(* PLC project SingleResponsibility.project, CODESYS CODESYS V3.5 SP10 Patch 4 *)
(* stored: creationDateTime 2017-07-22T20:32:32.9692432, modificationDateTime 2017-06-30T11:24:00.4798052 *)

INTERFACE IEStoppable
METHOD executeEStop
END_METHOD
END_INTERFACE

INTERFACE IRunnable
METHOD run
END_METHOD
END_INTERFACE

INTERFACE IStoppable
METHOD stop
END_METHOD
END_INTERFACE

INTERFACE IEdge
METHOD isRising : BOOL
END_METHOD
METHOD isFalling : BOOL
END_METHOD
END_INTERFACE

INTERFACE ISensor
METHOD isOccupied : BOOL
END_METHOD
METHOD isFree : BOOL
END_METHOD
END_INTERFACE

INTERFACE IReciverInterface
METHOD readExtCondition2Rec : IReciverInterface
  VAR_INPUT
    receiveCondition : BOOL;  (* condition 4 ready to receive *)
  END_VAR
END_METHOD
METHOD isReceiving : BOOL
END_METHOD
END_INTERFACE

INTERFACE ISenderInterface
METHOD readExtCondition2Snd : ISenderInterface
  VAR_INPUT
    sendCondition : BOOL;  (* condition 4 ready 2 send *)
  END_VAR
END_METHOD
METHOD isSending : BOOL
END_METHOD
END_INTERFACE

INTERFACE ISmema
METHOD setCondition
  VAR_INPUT
    smemaCondition : BOOL;  (* must be ture to activate the smema interface *)
  END_VAR
END_METHOD
METHOD isTransferActive : BOOL
END_METHOD
END_INTERFACE

INTERFACE ITwoStageLinearDrive
METHOD fastForward
END_METHOD
METHOD forward
END_METHOD
METHOD fastBackward
END_METHOD
METHOD backward
END_METHOD
END_INTERFACE

INTERFACE ITwoStageRotationDrive
METHOD fastClockwise
END_METHOD
METHOD clockwise
END_METHOD
METHOD fastCounterClockwise
END_METHOD
METHOD counterClockwise
END_METHOD
END_INTERFACE

INTERFACE IMachineState
METHOD isMachineInInitMode : BOOL
END_METHOD
METHOD isMachineInIdle : BOOL
END_METHOD
METHOD isMachineInSetup : BOOL
END_METHOD
METHOD isMachineInAutomatic : BOOL
END_METHOD
METHOD isMachineInEstop : BOOL
END_METHOD
END_INTERFACE

FUNCTION_BLOCK DebouncedDigitalSensor IMPLEMENTS ISensor, IEdge
  VAR
    diSensor : REFERENCE TO BOOL;  (* reference to the digital input *)
    maskOccupied : BOOL;  (* mask for the state occupied *)
    debouncer : TON;  (* ton to debounce the sensor signal *)
    debounceTime : TIME;  (* debounce time *)
    state : BOOL;  (* sensor state *)
  END_VAR

            
          

METHOD isOccupied : BOOL
                  isOccupied := isSensorInState(state := THIS^.maskOccupied);
                
END_METHOD

METHOD isFree : BOOL
                  isFree := isSensorInState(state := (NOT THIS^.maskOccupied));
                
END_METHOD

METHOD isRising : BOOL
                  isRising 	:= (THIS^.isOccupied() AND (NOT THIS^.state));
THIS^.updateState();
                
END_METHOD

METHOD isFalling : BOOL
                  isFalling 	:= (THIS^.isFree() AND THIS^.state);
THIS^.updateState();
                
END_METHOD

METHOD FB_INIT
  VAR_INPUT
    bInitRetains : BOOL;  (* initializing of retain-variable *)
    bInCopyCode : BOOL;  (* instance is copied to copy-code *)
    diSensor : REFERENCE TO BOOL;  (* reference to the digital input *)
    maskOccupied : BOOL;  (* mask for the state occupied *)
  END_VAR
                  THIS^.diSensor		REF=diSensor; 
THIS^.maskOccupied	:= maskOccupied;
THIS^.debounceTime	:= T#30ms;
THIS^.state			:= (THIS^.diSensor = THIS^.maskOccupied);
                
END_METHOD

METHOD isSensorInState : BOOL
  VAR_INPUT
    state : BOOL;  (* requeseted sensor state *)
  END_VAR
                  THIS^.debouncer(IN := (THIS^.diSensor = state), PT := THIS^.debounceTime, Q => isSensorInState);
                
END_METHOD

METHOD updateState
                  THIS^.state := THIS^.isOccupied();
                
END_METHOD
END_FUNCTION_BLOCK

FUNCTION_BLOCK SmemaInterface IMPLEMENTS ISmema
  VAR
    machineStateHndl : IMachineState;  (* machine state handler to check if receiving is allowed *)
    partnerIsRdy : REFERENCE TO BOOL;  (* ready signal from the interface partner *)
    weAreRdy : REFERENCE TO BOOL;  (* ready signal to the interface partner *)
    transferCondition : BOOL;  (* external condition for transfer is possible *)
    maskPartnerIsRdy : BOOL;  (* bitmask for partner is ready *)
    maskWeAreRdy : BOOL;  (* bitmask for we are ready *)
  END_VAR

            
          

METHOD setCondition
  VAR_INPUT
    smemaCondition : BOOL;  (* must be ture to activate the smema interface *)
  END_VAR
                  THIS^.transferCondition	:= transferCondition;
IF (NOT THIS^.transferCondition) THEN
	THIS^.weAreRdy := (NOT THIS^.maskWeAreRdy);
END_IF;
                
END_METHOD

METHOD isTransferActive : BOOL
                  IF (THIS^.transferCondition AND THIS^.machineStateHndl.isMachineInAutomatic()) THEN
	THIS^.weAreRdy := THIS^.maskWeAreRdy;
ELSE
	THIS^.weAreRdy := (NOT THIS^.maskWeAreRdy);
END_IF;		
isTransferActive	  := ((THIS^.weAreRdy = THIS^.maskWeAreRdy) AND (THIS^.maskPartnerIsRdy = THIS^.maskPartnerIsRdy));

                
END_METHOD

METHOD FB_INIT
  VAR_INPUT
    bInitRetains : BOOL;  (* initializing of retain-variable *)
    bInCopyCode : BOOL;  (* instance is copied to copy-code *)
    partnerIsRdy : REFERENCE TO BOOL;  (* ready signal from the interface partner *)
    weAreRdy : REFERENCE TO BOOL;  (* ready signal to the interface partner *)
    maskPartnerIsRdy : BOOL;  (* bitmask for partner is ready *)
    maskWeAreRdy : BOOL;  (* bitmask for we are ready *)
    machineStateHndl : IMachineState;  (* the machine is in machine state automatic *)
  END_VAR
                  THIS^.partnerIsRdy	    REF= partnerIsRdy;
THIS^.weAreRdy		    REF= weAreRdy;
THIS^.machineStateHndl	:= 	 machineStateHndl;
THIS^.transferCondition	:=	 FALSE;
THIS^.maskPartnerIsRdy	:=   maskPartnerIsRdy;
THIS^.maskWeAreRdy		:=	 maskWeAreRdy;
                
END_METHOD
END_FUNCTION_BLOCK

FUNCTION_BLOCK SmemaReceiver IMPLEMENTS IReciverInterface
  VAR
    smeaInterface : ISmema;  (* smema interface for the receiver *)
  END_VAR

            
          

METHOD isReceiving : BOOL
                  isReceiving	  := (THIS^.smeaInterface.isTransferActive());
                
END_METHOD

(* inject conditions for ready to receive *)
METHOD readExtCondition2Rec : IReciverInterface
  VAR_INPUT
    receiveCondition : BOOL;  (* condition 4 ready to receive *)
  END_VAR
                  THIS^.smeaInterface.setCondition(smemaCondition := receiveCondition);
readExtCondition2Rec	:= THIS^;
                
END_METHOD

METHOD FB_INIT
  VAR_INPUT
    bInitRetains : BOOL;  (* initializing of retain-variable *)
    bInCopyCode : BOOL;  (* instance is copied to copy-code *)
    smeaInterface : ISmema;  (* smema interface for the receiver *)
  END_VAR
                  THIS^.smeaInterface	:= 	 smeaInterface ;
                
END_METHOD
END_FUNCTION_BLOCK

FUNCTION_BLOCK SmemaSender IMPLEMENTS ISenderInterface
  VAR
    smeaInterface : ISmema;  (* smema interface for the sender *)
  END_VAR

            
          

(* inject conditions for ready to receive *)
METHOD readExtCondition2Snd : ISenderInterface
  VAR_INPUT
    sendCondition : BOOL;  (* condition 4 ready 2 send *)
  END_VAR
                  THIS^.smeaInterface.setCondition(smemaCondition := sendCondition);
readExtCondition2Snd := THIS^;
                
END_METHOD

METHOD isSending : BOOL
                  isSending	  := (THIS^.smeaInterface.isTransferActive());
                
END_METHOD

METHOD FB_INIT
  VAR_INPUT
    bInitRetains : BOOL;  (* initializing of retain-variable *)
    bInCopyCode : BOOL;  (* instance is copied to copy-code *)
    smeaInterface : ISmema;  (* smema interface for the sender *)
  END_VAR
                  THIS^.smeaInterface	:= 	 smeaInterface ;
                
END_METHOD
END_FUNCTION_BLOCK

FUNCTION_BLOCK Conveyor2ndTry IMPLEMENTS IRunnable
  VAR
    slowSensor : ISensor;  (* sensor to slow down *)
    stopSensor : ISensor;  (* sensor to stop *)
    senderInterface : ISenderInterface;  (* interface to send *)
    receiverInterface : IReciverInterface;  (* interface to receive *)
    drive : ITwoStageLinearDrive;  (* drive to run the conveyor *)
    machineState : IMachineState;  (* just the machine state *)
  END_VAR

            
          

METHOD run
                  (*recive part*)
IF (THIS^.receiverInterface.readExtCondition2Rec(receiveCondition := THIS^.isEmpty()).isReceiving()) THEN
	THIS^.drive.fastForward();
(*send part*)
ELSIF (THIS^.senderInterface.readExtCondition2Snd(sendCondition := (THIS^.isAligned() OR THIS^.isOccupiedOutfeed())).isSending()) THEN
	THIS^.drive.fastForward();
(*align part*)
ELSIF (THIS^.isOccupiedInfeed() AND THIS^.machineState.isMachineInAutomatic()) THEN
	THIS^.drive.forward();
ELSE
	THIS^.drive.stop();
END_IF
                
END_METHOD

METHOD FB_INIT
  VAR_INPUT
    bInitRetains : BOOL;  (* initializing of retain-variable *)
    bInCopyCode : BOOL;  (* instance is copied to copy-code *)
    slowSensor : ISensor;  (* sensor to slow down *)
    stopSensor : ISensor;  (* sensor to stop *)
    senderInterface : ISenderInterface;  (* interface to send *)
    receiverInterface : IReciverInterface;  (* interface to receive *)
    drive : ITwoStageLinearDrive;  (* drive to run the conveyor *)
    machineState : IMachineState;  (* just the machine state *)
  END_VAR
                  //sensors
THIS^.slowSensor	    := slowSensor; //sensor to slow down
THIS^.stopSensor	    := stopSensor; //sensor to stop
//interfaces
THIS^.senderInterface	:= senderInterface	; //interface to send
THIS^.receiverInterface	:= receiverInterface; //interface to receive
//conveyor drive
THIS^.drive 			:= drive; //drive to run the conveyor
//machine state
THIS^.machineState		:= machineState; //just the machine state
                
END_METHOD

METHOD isEmpty : BOOL
                  isEmpty := (THIS^.slowSensor.isFree() AND THIS^.stopSensor.isFree());
                
END_METHOD

METHOD isAligned : BOOL
                  isAligned := (THIS^.slowSensor.isOccupied() AND THIS^.stopSensor.isOccupied());
                
END_METHOD

METHOD isOccupiedInfeed : BOOL
                  isOccupiedInfeed := (THIS^.slowSensor.isOccupied() AND THIS^.stopSensor.isFree());
                
END_METHOD

METHOD isOccupiedOutfeed : BOOL
                  isOccupiedOutfeed := (THIS^.slowSensor.isFree() AND THIS^.stopSensor.isOccupied());
                
END_METHOD
END_FUNCTION_BLOCK

FUNCTION_BLOCK Acme2StageDrive EXTENDS ACommonTwoStageDrive
  VAR
    cw : REFERENCE TO BOOL;  (* run the motor clockwise, if it false the motor will run counter clockwise *)
    fast : REFERENCE TO BOOL;  (* run the motor fast, if it false will the motor running slow *)
    start : REFERENCE TO BOOL;  (* run start the motor *)
    maskFwd : BOOL;  (* mask to define forward or rather clockwise *)
  END_VAR

            
          

METHOD stop
                  THIS^.start := FALSE;
                
END_METHOD

METHOD fastForward
                  THIS^.StartMotor(direction := THIS^.maskFwd, velocity := TRUE);
                
END_METHOD

METHOD forward
                  THIS^.StartMotor(direction := THIS^.maskFwd, velocity := FALSE);
                
END_METHOD

METHOD fastBackward
                  THIS^.StartMotor(direction := (NOT THIS^.maskFwd), velocity := TRUE);
                
END_METHOD

METHOD backward
                  THIS^.StartMotor(direction := (NOT THIS^.maskFwd), velocity := FALSE);
                
END_METHOD

METHOD fastClockwise
                  THIS^.fastForward();
                
END_METHOD

METHOD clockwise
                  THIS^.forward();
                
END_METHOD

METHOD fastCounterClockwise
                  THIS^.fastBackward();
                
END_METHOD

METHOD counterClockwise
                  THIS^.backward();
                
END_METHOD

METHOD executeEStop
                  THIS^.stop();
                
END_METHOD

METHOD FB_INIT
  VAR_INPUT
    bInitRetains : BOOL;  (* initializing of retain-variable *)
    bInCopyCode : BOOL;  (* instance is copied to copy-code *)
    cw : REFERENCE TO BOOL;  (* run the motor clockwise, if it false the motor will run counter clockwise *)
    fast : REFERENCE TO BOOL;  (* run the motor fast, if it false will the motor running slow *)
    start : REFERENCE TO BOOL;  (* run start the motor *)
    maskFwd : BOOL;  (* mask to define forward or rather clockwise *)
  END_VAR
                  THIS^.cw             REF= cw ;
THIS^.fast           REF= fast ;
THIS^.start          REF= start ;
THIS^.maskFwd      	 :=   maskFwd;
                
END_METHOD

METHOD StartMotor
  VAR_INPUT
    direction : BOOL;  (* direction flag *)
    velocity : BOOL;  (* velocity flag *)
  END_VAR
                  THIS^.cw 	 	:= direction;
THIS^.fast   	:= velocity;
THIS^.start  	:= TRUE;
                
END_METHOD
END_FUNCTION_BLOCK

FUNCTION_BLOCK ACommonTwoStageDrive IMPLEMENTS ITwoStageLinearDrive, ITwoStageRotationDrive, IEStoppable

            
          

METHOD stop
                  
                
END_METHOD

METHOD fastForward
                  
                
END_METHOD

METHOD forward
                  
                
END_METHOD

METHOD fastBackward
                  
                
END_METHOD

METHOD backward
                  
                
END_METHOD

METHOD fastClockwise
                  
                
END_METHOD

METHOD clockwise
                  
                
END_METHOD

METHOD fastCounterClockwise
                  
                
END_METHOD

METHOD counterClockwise
                  
                
END_METHOD

METHOD executeEStop
                  
                
END_METHOD

METHOD FB_INIT
  VAR_INPUT
    bInitRetains : BOOL;  (* initializing of retain-variable *)
    bInCopyCode : BOOL;  (* instance is copied to copy-code *)
  END_VAR
                  
                
END_METHOD
END_FUNCTION_BLOCK

PROGRAM PLC_PRG

                    
                  
END_PROGRAM

CONFIGURATION Device
  RESOURCE Application ON PLC
    TASK MainTask(INTERVAL := T#20ms, PRIORITY := 1);
    PROGRAM PLC_PRG WITH MainTask : PLC_PRG;
  END_RESOURCE
END_CONFIGURATION
